TEXTLIST HandlingModulesCmd
  0 = 'NOP'
  10 = 'STOP'
  20 = 'RESET'
  60 = 'POWER'
  100 = 'HOME'
  300 = 'MAN'
  500 = 'LOAD'
  3000 = 'MOVE'
  800 = 'UNLOAD'
  1000 = 'DO'
   = ''
END_TEXTLIST

(* stored: Version 1.1.0.1, ProductVersion 3.1.4024.11
   TextList HandlingModulesCmd: Id {3744f94f-d6d0-4f39-83c0-c362b71844a4} *)
